(* CoDeSys 2.3.9.41 project: OWENProject.pro *)
(* Libraries: Util.lib 18.5.10 15:14:28, STANDARD.LIB 4.10.05 11:14:46, IECSFC.LIB 13.4.06 15:51:28, ANALYZATION.LIB 5.10.99 09:05:06 *)

(* PLC configuration (modules and I/O channels)
Fast discrete inputs [I_SIMPLE_INPUT] node 0, in %IB0 out %QB0 {Filtrationtime = 10}
  AT %IX0.0 [BitInput] Discrete input 1
  AT %IX0.1 [BitInput] Discrete input 2
  AT %IX0.2 [BitInput] Discrete input 3
  AT %IX0.3 [BitInput] Discrete input 4
Discrete inputs [ID130] node 1, in %IB1 out %QB1 {Filtrationtime_GeneralINP = 10; Visibility = No; PinCount = 12}
  AT %IB1.0 [ByteInput] 8 discrete inputs
  AT %IB1.1 [ByteInput] 4 discrete inputs
AT %QB2.0 [ByteOutput] 8 discrete outputs
AT %QB2.1 [ByteOutput] 4 discrete outputs
AT %IR3.0 [FloatInputP] AI #1 {AIN_TYPE = 4-20 mA; Peak_Filtr = 200; Flt_Ch = Off; TauRC = 10; MinFV = 0; MaxFV = 50}
AT %IR3.1 [FloatInputP] AI #2 {AIN_TYPE = 4-20 mA; Peak_Filtr = 200; Flt_Ch = Off; TauRC = 10; MinFV = 0; MaxFV = 50}
AT %IR3.2 [FloatInputP] AI #3 {AIN_TYPE = 4-20 mA; Peak_Filtr = 200; Flt_Ch = Off; TauRC = 10; MinFV = 0; MaxFV = 50}
AT %IR3.3 [FloatInputP] AI #4 {AIN_TYPE = 4-20 mA; Peak_Filtr = 200; Flt_Ch = Off; TauRC = 10; MinFV = 0; MaxFV = 20000.0}
AT %IR3.4 [FloatInputP] AI #5 {AIN_TYPE = 4-20 mA; Peak_Filtr = 200; Flt_Ch = Off; TauRC = 10; MinFV = 0; MaxFV = 20000.0}
AT %IR3.5 [FloatInputP] AI #6 {AIN_TYPE = 4-20 mA; Peak_Filtr = 200; Flt_Ch = Off; TauRC = 10; MinFV = 0; MaxFV = 20000.0}
AT %IR3.6 [FloatInputP] AI #7 {AIN_TYPE = 4-20 mA; Peak_Filtr = 200; Flt_Ch = Off; TauRC = 10; MinFV = 0; MaxFV = 20000.0}
AT %IR3.7 [FloatInputP] AI #8 {AIN_TYPE = 4-20 mA; Peak_Filtr = 200; Flt_Ch = Off; TauRC = 10; MinFV = 0; MaxFV = 20000.0}
AT %IW3.8 [WordInput] AI read time (10ms)
AT %QR4.0 [FloatOutputP] AO #1 {AOUT_TYPE = 0-10V; SafeValueREAL = 0.0}
AT %QR4.1 [FloatOutputP] AO #2 {AOUT_TYPE = 0-10V; SafeValueREAL = 0.0}
AT %QR4.2 [FloatOutputP] AO #3 {AOUT_TYPE = 0-10V; SafeValueREAL = 0.0}
AT %QR4.3 [FloatOutputP] AO #4 {AOUT_TYPE = 4-20 mA; SafeValueREAL = 0.0}
Special input [ID103] node 5, in %IB5 out %QB5 {Filtrationtime = 1000; PinCount = 1; WatchDogPeriod = 400; PollPeriod = 3000; Visibility = No}
  AT %IX5.0 [BitInput] Special input
Special output [ID104] node 6, in %IB6 out %QB6 {Visibility = No; PinCount = 1}
  AT %QX6.0 [BitOutput] Special output
Owen (Master) [OWEN_MASTER_ID451] node 7, in %IB7 out %QB7 {Timeout = 50; Visibility = Yes}
  AT %QW7.0 [WordOutput] Last error
  AT %QW7.1 [WordOutput] Last hash
  AT %QW7.2 [WordOutput] Last address
  AT %QB7.3 [ComChannel] Start/Stop)
  RS-485-1 [COM1_USART] node 0, in %IB7.0 out %QB7.0 {CommunicationSpeed = 9600; Parity = NO PARITY CHECK; BitLength = 8 bits; StopLength = One stop bit; InterfaceType = RS485; FrameOriented = ASCII; Timeout = 2; Visibility = No}
AT %QD7.1.0.0 [DWordOutput] MV110-32DN Digital Inputs
ModBus (Master) [MODBUS_MASTER_ID450] node 8, in %IB8 out %QB8 {Visibility = No}
  AT %QD8.0 [DWordOutput] Last address
  AT %QW8.1 [WordOutput] Last error
  RS-485-1 [COM1_USART] node 0, in %IB8.0 out %QB8.0 {CommunicationSpeed = 9600; Parity = NO PARITY CHECK; BitLength = 8 bits; StopLength = One stop bit; InterfaceType = RS485; FrameOriented = RTU; Timeout = 0; Visibility = No}
AT %QB8.1.0 [ComChannel] Command (0xff - Start)
AT %QW8.1.0.0 [WordOutput]
AT %QW8.1.1.0 [WordOutput]
AT %QW8.1.2.0 [WordOutput]
Value on output 4 [ID2085] node 3, in %IB8.1.3 out %QB8.1.3 {ModbusAddress = 3; Comm_Write_16 = Command Write (16); Visibility = No}
  AT %QW8.1.3.0 [WordOutput]
Value on output 5 [ID2086] node 4, in %IB8.1.4 out %QB8.1.4 {ModbusAddress = 4; Comm_Write_16 = Command Write (16); Visibility = No}
  AT %QW8.1.4.0 [WordOutput]
Value on output 6 [ID2087] node 5, in %IB8.1.5 out %QB8.1.5 {ModbusAddress = 5; Comm_Write_16 = Command Write (16); Visibility = No}
  AT %QW8.1.5.0 [WordOutput]
Value on output 7 [ID2088] node 6, in %IB8.1.6 out %QB8.1.6 {ModbusAddress = 6; Comm_Write_16 = Command Write (16); Visibility = No}
  AT %QW8.1.6.0 [WordOutput]
Value on output 8 [ID2089] node 7, in %IB8.1.7 out %QB8.1.7 {ModbusAddress = 7; Comm_Write_16 = Command Write (16); Visibility = No}
  AT %QW8.1.7.0 [WordOutput]
PWM period on output 1 [ID2090] node 8, in %IB8.1.8 out %QB8.1.8 {ModbusAddress = 32; Comm_Write_16 = Command Write (16); Visibility = No}
  AT %QW8.1.8.0 [WordOutput]
PWM period on output 2 [ID2091] node 9, in %IB8.1.9 out %QB8.1.9 {ModbusAddress = 33; Comm_Write_16 = Command Write (16); Visibility = No}
  AT %QW8.1.9.0 [WordOutput]
PWM period on output 3 [ID2092] node 10, in %IB8.1.10 out %QB8.1.10 {ModbusAddress = 34; Comm_Write_16 = Command Write (16); Visibility = No}
  AT %QW8.1.10.0 [WordOutput]
PWM period on output 4 [ID2093] node 11, in %IB8.1.11 out %QB8.1.11 {ModbusAddress = 35; Comm_Write_16 = Command Write (16); Visibility = No}
  AT %QW8.1.11.0 [WordOutput]
PWM period on output 5 [ID2094] node 12, in %IB8.1.12 out %QB8.1.12 {ModbusAddress = 36; Comm_Write_16 = Command Write (16); Visibility = No}
  AT %QW8.1.12.0 [WordOutput]
PWM period on output 6 [ID2095] node 13, in %IB8.1.13 out %QB8.1.13 {ModbusAddress = 37; Comm_Write_16 = Command Write (16); Visibility = No}
  AT %QW8.1.13.0 [WordOutput]
PWM period on output 7 [ID2096] node 14, in %IB8.1.14 out %QB8.1.14 {ModbusAddress = 38; Comm_Write_16 = Command Write (16); Visibility = No}
  AT %QW8.1.14.0 [WordOutput]
PWM period on output 8 [ID2097] node 15, in %IB8.1.15 out %QB8.1.15 {ModbusAddress = 39; Comm_Write_16 = Command Write (16); Visibility = No}
  AT %QW8.1.15.0 [WordOutput]
*)

(* Task configuration *)
TASK TaskFreewheeling (PRIORITY := 1); (* freewheeling *)
	PLC_PRG();
END_TASK
TASK Task200ms (PRIORITY := 1, INTERVAL := T#200ms);
	GetInputs();
END_TASK
TASK Task1Sec (PRIORITY := 1, INTERVAL := T#1000ms);
	SetOutputs();
END_TASK

(* Global variable list: Global_Variables *)
VAR_GLOBAL CONSTANT
	MAXIMUM_HEATING_CIRCUITS_NUM : USINT := 3;
	(*Количество отопительных контуров*)

	MAX_UZ_NUM : USINT := 3;
	(*Количество частотных преобразователей UZ*)

	MAX_BOILERS_NUM : USINT := 3;
	(*Количество котлов*)

	MAX_K14_PUMPS_NUM : USINT := 3;
	(*Количество насосов К14*)

	MAX_K15_PUMPS_NUM : USINT := 2;
	(*Количество насосов К15*)

	MAX_K16_PUMPS_NUM : USINT := 2;
	(*Количество насосов К16*)
END_VAR

VAR_GLOBAL
	PLC160DI : strPLC160DI;
	PLC160AI : strPLC160AI;
	PLC160DO : strPLC160DO;
	PLC160AO : strPLC160AO;
	MV110DI  : strMV110DI;
	MU110DO  : strMU110DO;

	K14PumpFaulty : ARRAY [1..MAX_K14_PUMPS_NUM] OF BOOL;
	(*Неиправен 1-3 насос группы К14?*)

	K15PumpFaulty : ARRAY [1..MAX_K15_PUMPS_NUM] OF BOOL;
	(*Неиправен 1-3 насос группы К16?*)

	K16PumpFaulty : ARRAY [1..MAX_K16_PUMPS_NUM] OF BOOL;
	(*Неиправен 1-3 насос группы К16?*)
END_VAR

(* Global variable list: PLC_IO *)
VAR_GLOBAL
(* Дискретные входы ПЛК160*)
	DI_0_00  AT %IX0.0 : BOOL;
	DI_0_01  AT %IX0.1 : BOOL;
	DI_0_02  AT %IX0.2 : BOOL;
	DI_0_03  AT %IX0.3 : BOOL;
	DI_0_04  AT %IX1.0.0 : BOOL;
	DI_0_05  AT %IX1.0.1 : BOOL;
	DI_0_06  AT %IX1.0.2 : BOOL;
	DI_0_07  AT %IX1.0.3 : BOOL;
	DI_0_08  AT %IX1.0.4 : BOOL;
	DI_0_09  AT %IX1.0.5 : BOOL;
	DI_0_10  AT %IX1.0.6 : BOOL;
	DI_0_11  AT %IX1.0.7 : BOOL;
	DI_0_12  AT %IX1.1.0 : BOOL;
	DI_0_13  AT %IX1.1.1 : BOOL;
	DI_0_14  AT %IX1.1.2 : BOOL;
	DI_0_15  AT %IX1.1.3 : BOOL;

(* Аналоговые входы ПЛК160*)
	AI_0_00 AT %IR3.0 : REAL;
	AI_0_01 AT %IR3.1 : REAL;
	AI_0_02 AT %IR3.2 : REAL;
	AI_0_03 AT %IR3.3 : REAL;
	AI_0_04 AT %IR3.4 : REAL;
	AI_0_05 AT %IR3.5 : REAL;
	AI_0_06 AT %IR3.6 : REAL;
	AI_0_07 AT %IR3.7 : REAL;

(*Аналоговые выходы ПЛК160*)
	AO_0_00 AT %QR4.0 : REAL;
	AO_0_01 AT %QR4.1 : REAL;
	AO_0_02 AT %QR4.2 : REAL;
	AO_0_03 AT %QR4.3 : REAL;

(*Дискретные выходы ПЛК160*)
	DO_0_00 AT %QX2.0.0 : BOOL;
	DO_0_01 AT %QX2.0.1 : BOOL;
	DO_0_02 AT %QX2.0.2 : BOOL;
	DO_0_03 AT %QX2.0.3 : BOOL;
	DO_0_04 AT %QX2.0.4 : BOOL;
	DO_0_05 AT %QX2.0.5 : BOOL;
	DO_0_06 AT %QX2.0.6 : BOOL;
	DO_0_07 AT %QX2.0.7 : BOOL;

	DO_0_08 AT %QX2.1.0 : BOOL;
	DO_0_09 AT %QX2.1.1 : BOOL;
	DO_0_10 AT %QX2.1.2 : BOOL;
	DO_0_11 AT %QX2.1.3 : BOOL;

(*Дискретные входы МВ110-32ДН*)
	DI_1 AT %QD7.1.0.0 : DWORD;

(*Дискретные выходы МУ110-8Р*)
	DO_1_00 AT %QW8.1.0.0 : WORD;
	DO_1_01 AT %QW8.1.1.0 : WORD;
	DO_1_02 AT %QW8.1.2.0 : WORD;
	DO_1_03 AT %QW8.1.3.0 : WORD;
	DO_1_04 AT %QW8.1.4.0 : WORD;
	DO_1_05 AT %QW8.1.5.0 : WORD;
	DO_1_06 AT %QW8.1.6.0 : WORD;
	DO_1_07 AT %QW8.1.7.0 : WORD;


END_VAR

(* Global variable list: Variable_Configuration *)
VAR_GLOBAL RETAIN
	K14UZSPumpSpeed : USINT := 100;
END_VAR

(* Data type *)
TYPE strMU110DO :
STRUCT
	K14PumpGroupAlarm : BOOL;
(*
	Выход №1
	Авария насосной группы К14
*)

	Buzzer : BOOL;
(*
	Выход №2
	Зуммер
*)

	K14PumpIsOn : ARRAY [1..MAX_K14_PUMPS_NUM] OF BOOL;
(*
	Выходы №3-5
	"Насос К14.1-3 в работе"
*)

	Reserved : ARRAY [1..3] OF BOOL;
(*
	Выходы 6-8
	Резерв
*)


END_STRUCT
END_TYPE

(* Data type *)
TYPE strMV110DI :
(*
	поз. А2
	Контроллер МВ110-32 ДН
	Дискретные входы
*)
STRUCT
	K15_StopButton : ARRAY [1..2] OF BOOL;
(*
	Входы №1-2
	Сигналы с кнопок стоп Насосов К15.1-2
*)

	K16_StopButton : ARRAY [1..2] OF BOOL;
(*
	Входы №3-4
	Сигналы с кнопок стоп Насосов К16.1-2
*)

	K15_NoPressureDrop : BOOL;
(*
	Вход №5
	Сигнал с датчика перепада давления
	"Нет перепада давления на насосной группе К15"
	Замкнут - "Нет перепада".
*)

	K16_NoPressureDrop : BOOL;
(*
	Вход №6
	Сигнал с датчика перепада давления
	"Нет перепада давления на насосной группе К16"
	Замкнут - "Нет перепада".
*)

	HeatingDHWPumpGroupModeIsAuto : BOOL;
(*
	Вход №7
	Сигнал переключателя "Работа в автоматическом режиме
	насосной группы К15 греющего контура ГВС"
*)

	DHWPumpGroupModeIsAuto : BOOL;
(*
	Вход №8
	Сигнал переключателя "Работа в автоматическом режиме
	насосной группы К16 контура ГВС"
*)

	CO_Level_I : BOOL;
(*
	Вход №9
	I уровень загазованности по CO
*)

	CO_Level_II : BOOL;
(*
	Вход №10
	II уровень загазованности по CO
*)

	CH_Level_I : BOOL;
(*
	Вход №11
	I уровень загазованности по CH
*)

	CH_Level_II : BOOL;
(*
	Вход №12
	II уровень загазованности по CH
*)

	FireAlarm : BOOL;
(*
	Вход №13
	Пожар в энергоцентре
*)

	BoilerGeneralFault : BOOL;
(*
	Вход №14
	Сигнал с панели управления котлов ведущей ПУКВ
	"Общая неисправность котлов"
*)

	TurnOnK15AndK16 : BOOL;
(*
	Вход №15
	Сигнал с панели управления котлов ведущей ПУКВ,
	"Включить/Выключить насосную группу К15 и К16"
*)

	K22ValveState : strValveState;
(*
	Входы №16-17
	Сигналы положения 3-х ходового клапана К22 "Открыт"/"Закрыт"
*)

	K23ValveState : strValveState;
(*
	Входы №18-19
	Сигналы положения 3-х ходового клапана К23 "Открыт"/"Закрыт"
*)

	BoilerAlarm : ARRAY [1..MAX_BOILERS_NUM] OF BOOL;
(*
	Входы №20-22
	Сигналы с ЩАК1-3 "Авария котла №1-3"
*)

	BlockAllBoilers : BOOL;
(*
	Вход №23
	Блокировка всех котлов
*)

	TurnOnAllBoilers : BOOL;
(*
	Вход №24
	Сигнал внешнего включения всех котлов
*)

	SignalizationButton : BOOL;
(*
	Вход №25
	Кнопка съема сигнализации
*)

	QFSwitcher : ARRAY [1..7] OF BOOL;
(*
	Входы №26-32
	Доп. контакты автоматических выключателей QF1-7
	1-3 Включение/выключение частотных модуляторов UZ
	4-5 - Включение/выключение насосов К15
	6-7 - Включение/выключение насосов К16
*)


END_STRUCT
END_TYPE

(* Data type *)
TYPE strPLC160AI :
(*
	поз. А1
	Контроллер ПЛК160
	Аналоговые входы
*)
STRUCT
	UZSignal : ARRAY [1..MAX_UZ_NUM] OF tUZSignal;
(*
	Аналоговые входы №1-3:
	Сигналы 0-20mA от частотных преобразователей UZ
*)

	DilutionSignal : ARRAY [1..MAX_BOILERS_NUM] OF tDelutionSignal;
(*
	Аналоговые входы №4-6:
	Сигналы 4-20mA измерения разрежения из щита ЩИР
	по одному сигналу на каждый котел
*)

	Reserved : ARRAY [1..2] OF tAnalogInput;
(*
	Незадействованные входы
*)


END_STRUCT
END_TYPE

(* Data type *)
(*
	поз. А1
	Контроллер ПЛК160
	Аналоговые выходы
*)
TYPE strPLC160AO :
STRUCT
(*
	Выходы №1-3
	Задание частоты для UZ1-3
	Сигнал 0-10V
*)
	UZSpeed : ARRAY [1..MAX_UZ_NUM] OF tUZSpeed;

(*
	Выход №4
	Резерв
*)
	Reserved : tAnalogOutput;
END_STRUCT
END_TYPE

(* Data type *)
TYPE strPLC160DI :
STRUCT
	K14_PumpsModeIsAuto : BOOL;
(*
	Дискретных вход №1:
	Сигнал с переключателя режима работы насосов К14
	"Ручной/Автоматический". Замкнут - "Автоматический"
*)

	K14_PumpsModeIsHeating : BOOL;
(*
	Дискретный вход №2:
	Сигнал с переключателя режима работы насосов К14
	"Летний/Отопительный". Замкнут - "Отопительный"
*)

	K14_PumpStop : ARRAY [1..MAX_K14_PUMPS_NUM] OF BOOL;
(*
	Дискретный вход №3-5:
	Сигнал с кнопки "Стоп насос К14.1-3".
	Замкнут - "Кнопка нажата".
	Аварийный СТОП насоса
*)

	K14_NoPressureDrop : BOOL;
(*
	Дискретный вход №6:
	Сигнал с датчика перепада давления
	насосной группы К14.
	Замкнут - нет перепада.
*)

	UZStatus : ARRAY [1..MAX_UZ_NUM] OF strUZStatus;
(*
	Дискретные входы №7-15:
	Сигналы част. преобр. UZ1-UZ3
*)

	Reserved : BOOL;
(*
	Дискретный вход №16:
	Резерв
*)


END_STRUCT
END_TYPE

(* Data type *)
TYPE strPLC160DO :
(*
	поз. А1
	Контроллер ПЛК160
	Дискретные выходы
*)
STRUCT
	UZStart : ARRAY [1..MAX_UZ_NUM] OF BOOL;
(*
	Выходы №1-3
	Пуск UZ
*)

	UZConstSpeed : ARRAY [1..MAX_UZ_NUM] OF BOOL;
(*
	Выходы №4-6
	Выбор постоянной скорости UZ (50Гц, 100%)
*)

	K15Pump : ARRAY [1..2] OF BOOL;
(*
	Выходы №7-8
	Включить/отключить насосы К15.1-2
*)

	K16Pump : ARRAY [1..2] OF BOOL;
(*
	Выходы №9-10
	Включить/отключить насосы К16.1-2
*)

	K15Alarm : BOOL;
(*
	Выход №11
	Авария насосной группы К15
*)

	K16Alarm : BOOL;
(*
	Выход №12
	Авария насосной группы К16
*)



END_STRUCT
END_TYPE

(* Data type *)
(*Сигналы с част. преобр UZ*)
TYPE strUZStatus :
STRUCT
	Ready : BOOL;
	Running : BOOL;
	Fail	: BOOL;
END_STRUCT
END_TYPE

(* Data type *)
(*Состояние 3-х ходового клапана*)
TYPE strValveState :
STRUCT
	Open : BOOL;
	Close: BOOL;
END_STRUCT
END_TYPE

(* Data type *)
TYPE tAnalogInput : REAL;
END_TYPE

(* Data type *)
TYPE tAnalogOutput : REAL;
END_TYPE

(* Data type *)
TYPE tDelutionSignal : REAL;
END_TYPE

(* Data type *)
TYPE tUZSignal : REAL;
END_TYPE

(* Data type *)
TYPE tUZSpeed : REAL;
END_TYPE

(* POU PLC_PRG, ST *)
PROGRAM PLC_PRG
VAR CONSTANT
	K14AutoModeDelay : TIME := T#10s;
END_VAR

VAR
	SignalizationResetTrigger : F_TRIG;
	K14PumpsControl : fbK14PumpsControl;
	K15PumpsControl : fbK15PumpsControl;
	K16PumpsControl : fbK16PumpsControl;
	K14ManualModeTOF : TOF;
END_VAR

VAR_TEMP
	i: USINT;
	K14WorkAllowed : BOOL := FALSE;

	K15WorkAllowed: BOOL := FALSE;

	K16WorkAllowed : BOOL := FALSE;
END_VAR
	K14WorkAllowed := FALSE;

	K15WorkAllowed := FALSE;

	K16WorkAllowed := FALSE;

(*
	Проверить состояние аварий на насосах и зажечь лампочки, включить зуммер
*)
checkPumpsAlarm();

(*
	Проверить состояние всех других аварий и включить зуммер
*)
checkOtherAlarms();

(*
	Сброс всех аварий насосов по замыканию кнопки
	съема аварий
*)
SignalizationResetTrigger(CLK := MV110DI.SignalizationButton);
resetPumpsAlarm(SignalizationResetTrigger.Q);


(*
	Включение сигнала на UZ
	по тому же сигналу, что и MV110DI.TurnOnK15AndK16
FOR i := 1 TO MAX_K14_PUMPS_NUM DO
	PLC160DO.UZStart[i] := MV110DI.TurnOnK15AndK16;
END_FOR;
*)

(*
	3. Управление насосами К14
	контура отопления и вентиляции
*)
FOR i := 1 TO MAX_K14_PUMPS_NUM DO
	MU110DO.K14PumpIsOn[i] := PLC160DI.UZStatus[i].Running;
	(*Включить/Выключить сигнальную лампу состояния насоса*)

	(*если хоть один из насосов исправен, то работа разрешена*)
	IF NOT(K14PumpFaulty[i]) THEN
		K14WorkAllowed := TRUE;
	END_IF;
END_FOR;

K14ManualModeTOF(IN := NOT(PLC160DI.K14_PumpsModeIsAuto), PT := K14AutoModeDelay);

K14PumpsControl(
	ManualMode						:= K14ManualModeTOF.Q,
	WorkAllowed						:= K14WorkAllowed,
	SummerMode						:= NOT(PLC160DI.K14_PumpsModeIsHeating),
	EmergencyPumpStopButtonPressed := PLC160DI.K14_PumpStop,
	PumpState						:= MU110DO.K14PumpIsOn,
	PressureDrop					:= NOT(PLC160DI.K14_NoPressureDrop)
);

(*
	6. Управление насосами К15
	греющего контура ГВС
*)
FOR i := 1 TO MAX_K15_PUMPS_NUM DO
	(*если хоть один из насосов исправен, то работа разрешена*)
	IF NOT(K15PumpFaulty[i]) THEN
		K15WorkAllowed := TRUE;
	END_IF;
END_FOR;

K15PumpsControl(
	ManualMode						:= NOT(MV110DI.HeatingDHWPumpGroupModeIsAuto),
	WorkAllowed						:= K15WorkAllowed,
	EmergencyPumpStopButtonPressed := MV110DI.K15_StopButton,
	PumpState						:= PLC160DO.K15Pump,
	PressureDrop					:= NOT(MV110DI.K15_NoPressureDrop)
);

(*
	5. Управление насосами К16
	контура ГВС
*)
FOR i := 1 TO MAX_K16_PUMPS_NUM DO
	(*если хоть один из насосов исправен, то работа разрешена*)
	IF NOT(K16PumpFaulty[i]) THEN
		K16WorkAllowed := TRUE;
	END_IF;
END_FOR;

K16PumpsControl(
	ManualMode						:= NOT(MV110DI.DHWPumpGroupModeIsAuto),
	WorkAllowed						:= K16WorkAllowed,
	EmergencyPumpStopButtonPressed := MV110DI.K16_StopButton,
	PumpState						:= PLC160DO.K16Pump,
	PressureDrop					:= NOT(MV110DI.K16_NoPressureDrop)
);
END_PROGRAM

(* POU K14/fbK14PumpsControl, ST *)
FUNCTION_BLOCK fbK14PumpsControl
(*
	3. Управление насосами К14
	контура отопления и вентиляции
*)
VAR CONSTANT
	PumpCheckDelayTime : TIME := T#30s;
END_VAR

VAR_INPUT
	ManualMode: BOOL;						(*Ручной режим?*)
	WorkAllowed: BOOL;					(*Работа разрешена?*)
	SummerMode: BOOL;						(*Летний режим?*)
	EmergencyPumpStopButtonPressed: ARRAY [1..MAX_K14_PUMPS_NUM] OF BOOL; (*Нажат аварийный стоп насоса?*)
	PumpState: ARRAY [1..MAX_K14_PUMPS_NUM] OF BOOL;	(*Работает насос?*)
	PressureDrop : BOOL;					(*Есть разница давлений?*)
END_VAR
VAR
	pumpStatusCheckDelay	: ARRAY [1..MAX_K14_PUMPS_NUM] OF TON;
	workOrderControl : fbK14WorkOrderControl;
	pumpsTrainingControl : fbK14PumpsTraining;
END_VAR
VAR_TEMP
	i: USINT;
	pumpWorkOrder : ARRAY [1..MAX_K14_PUMPS_NUM] OF USINT;
	pumpStatusCheck : ARRAY [1..MAX_K14_PUMPS_NUM] OF BOOL;
	break : BOOL := FALSE;
END_VAR
break := FALSE;
(*Проверяем исправность насосов К14*)
FOR i := 1 TO MAX_K14_PUMPS_NUM DO
	pumpStatusCheckDelay[i](IN := PumpState[i], PT := PumpCheckDelayTime);
	pumpStatusCheck[i] := pumpStatusCheckDelay[i].Q;
END_FOR;

fK14PumpsFaultyControl(
	PumpState				:= PumpState,
	PumpStatusCheckDelay	:= pumpStatusCheck,
	PressureDrop			:= PressureDrop
);

(*Управление насосами К14*)
IF ManualMode THEN (*Ручной режим?*)
(*
	FOR i := 1 TO MAX_K14_PUMPS_NUM DO
		fK14PumpManualControl(
			PumpID	:= i,
			TurnOn	:= TurnOnPumpButtonPressed[i],
			TurnOff	:= TurnOffPumpButtonPressed[i],
			State		:= PumpState[i],
			EmergencyStop := EmergencyPumpStopButtonPressed[i]
		);
	END_FOR;
*)
	(*Контроллер никак не участвует в ручном режиме*)
	FOR i := 1 TO MAX_K14_PUMPS_NUM DO
		fTurnOffK14Pump(i);
	END_FOR;
ELSE
	IF WorkAllowed THEN	(*Работа разрешена?*)
		(*определяем порядок включения насосов*)
		workOrderControl( SummerMode := SummerMode,
								pumpWorkOrder := pumpWorkOrder);

		FOR i := 1 TO MAX_K14_PUMPS_NUM DO
			(*
				работаем с насосами в порядке их приоритета
				Ищем первый исправный насос и включаем его
			*)
			IF NOT(break) AND NOT(K14PumpFaulty[pumpWorkOrder[i]]) THEN
				fK14PumpAutoControl(
						PumpID := pumpWorkOrder[i],
						EmergencyPumpStopButtonPressed := EmergencyPumpStopButtonPressed[pumpWorkOrder[i]]
				);
				break := TRUE;
			END_IF;
		END_FOR;
		(*периодическая тренировка насосов*)
		pumpsTrainingControl();
	ELSE
		(*
			если работа не разрешена,
			выключаем все насосы
		*)
		FOR i := 1 TO MAX_K14_PUMPS_NUM DO
			fTurnOffK14Pump(i);
		END_FOR;
		RETURN;
	END_IF;
END_IF;
END_FUNCTION_BLOCK

(* POU K14/fbK14WorkOrderControl, ST *)
FUNCTION_BLOCK fbK14WorkOrderControl
VAR_INPUT
	SummerMode: BOOL;
END_VAR

VAR CONSTANT
	MAX_K14_HEATING_ORDERS_NUM : USINT := 2;
	PumpWorkSummerOrder : ARRAY [1..MAX_K14_PUMPS_NUM] OF USINT := 3, 1, 2;
	PumpWorkHeatingOrder : ARRAY [1..MAX_K14_HEATING_ORDERS_NUM,
											1..MAX_K14_PUMPS_NUM] OF USINT := 1, 2, 3, 2, 1, 3;
END_VAR
VAR
	workOrderChanger		: BLINK;
	K14PumpsHeatingWorkOrderID : USINT(1..MAX_K14_HEATING_ORDERS_NUM) := 1;
END_VAR
VAR_IN_OUT
	pumpWorkOrder : ARRAY [1..MAX_K14_PUMPS_NUM] OF USINT;
END_VAR
VAR_TEMP
	i: USINT;
END_VAR
IF SummerMode THEN	(*Летний режим?*)
	pumpWorkOrder := PumpWorkSummerOrder;
ELSE

	workOrderChanger(
		ENABLE := TRUE,
		TIMELOW := T#24h,
		TIMEHIGH := T#24h
	);

	IF workOrderChanger.OUT THEN
		K14PumpsHeatingWorkOrderID := 1;
	ELSE
		K14PumpsHeatingWorkOrderID := 2;
	END_IF;

	FOR i := 1 TO MAX_K14_PUMPS_NUM DO
		pumpWorkOrder[i] := PumpWorkHeatingOrder[K14PumpsHeatingWorkOrderID, i];
	END_FOR;
END_IF;
END_FUNCTION_BLOCK

(* POU K14/fbK14PumpsTraining, ST *)
FUNCTION_BLOCK fbK14PumpsTraining
(*
	Функция тренировки насосов К14
*)
VAR CONSTANT
	TrainingDelay: TIME := T#24h;		(*Задержка на включение тренировки*)
	TrainingPeriod: TIME := T#10s;	(*Период тренировки*)
END_VAR
VAR
	PumpOffDelay : ARRAY [1..MAX_K14_PUMPS_NUM] OF TON;
	PumpTrainingTimer : ARRAY [1..MAX_K14_PUMPS_NUM] OF TP;
END_VAR
VAR_TEMP
	i: USINT;
END_VAR
FOR i := 1 TO MAX_K14_PUMPS_NUM DO
	PumpOffDelay[i](IN := fGetK14Pump(i), PT := TrainingDelay);
	PumpTrainingTimer[i](IN := PumpOffDelay[i].Q, PT := TrainingPeriod);
	IF PumpTrainingTimer[i].Q THEN
		fTurnOnK14Pump(i);
	END_IF;
END_FOR;
END_FUNCTION_BLOCK

(* POU K14/fGetK14Pump, ST *)
FUNCTION fGetK14Pump :BOOL
(* Проверка включения насоса*)
VAR_INPUT
	PumpID : USINT;
END_VAR
fGetK14Pump := MU110DO.K14PumpIsOn[PumpID];
END_FUNCTION

(* POU K14/fTurnOnK14Pump, ST *)
FUNCTION fTurnOnK14Pump : BOOL
VAR_INPUT
	PumpID : USINT;
END_VAR
VAR
END_VAR
	fSetK14Pump(TRUE, PumpID);
END_FUNCTION

(* POU K14/fSetK14Pump, ST *)
FUNCTION fSetK14Pump : BOOL
VAR_INPUT
	State	: BOOL;
	PumpID : USINT;
END_VAR
VAR
END_VAR
	(*Задать управляющее напряжение на насос*)
	IF State THEN
		PLC160DO.UZStart[PumpID]		:= TRUE;
		PLC160AO.UZSpeed[PumpID]	:= fUZSignalToVoltageOutput(K14UZSPumpSpeed);
	ELSE
		PLC160DO.UZStart[PumpID]		:= FALSE;
		PLC160AO.UZSpeed[PumpID]	:= 0.0;
	END_IF;
END_FUNCTION

(* POU K14/fUZSignalToVoltageOutput, ST *)
FUNCTION fUZSignalToVoltageOutput : REAL
(*
	Функция преобразования входного
	сигнала 0-100% в выходное управляющее
	напряжение на насос
*)
VAR_INPUT
	IN : USINT; (*Входной сигнал*)
END_VAR
VAR
END_VAR
(*TODO: написать корректную функцию преобразования тока в напряжение*)
fUZSignalToVoltageOutput := IN/10.0;
END_FUNCTION

(* POU K14/fK14PumpsFaultyControl, ST *)
FUNCTION fK14PumpsFaultyControl : BOOL
(* Проверка состояния насосов*)
VAR_INPUT
	PumpState : ARRAY [1..MAX_K14_PUMPS_NUM] OF BOOL;
	PumpStatusCheckDelay : ARRAY [1..MAX_K14_PUMPS_NUM] OF BOOL;
	PressureDrop : BOOL;
END_VAR
VAR
	i : USINT;
	activePumpID : USINT; (*номер работающего насоса*)
END_VAR
activePumpID := 0;

FOR i := 1 TO MAX_K14_PUMPS_NUM DO
	IF PumpState[i] THEN
		IF activePumpID <> 0 THEN
			(*
				Включено больше одного насоса -
				ничего не можем сказать об их исправности
			*)
			RETURN;
		END_IF;
		activePumpID := i;
	END_IF;
END_FOR;

IF activePumpID = 0 THEN
	(*
		Не включен ни один насос - 
		ничего не можем сказать об их исправности
	*)
	RETURN;
END_IF;

IF PumpStatusCheckDelay[activePumpID] THEN
	(*
		Определяем исправность насоса
		по перепаду давления
	*)
	K14PumpFaulty[activePumpID] := NOT(PressureDrop);
END_IF;
END_FUNCTION

(* POU K14/fTurnOffK14Pump, ST *)
FUNCTION fTurnOffK14Pump : BOOL
VAR_INPUT
	PumpID : USINT;
END_VAR
VAR
END_VAR
	fSetK14Pump(FALSE, PumpID);
END_FUNCTION

(* POU K14/fK14PumpAutoControl, ST *)
FUNCTION fK14PumpAutoControl : BOOL
VAR_INPUT
	PumpID : USINT;
	EmergencyPumpStopButtonPressed : BOOL;
END_VAR
VAR
	i : USINT;
END_VAR
(*выключаем все насосы кроме данного*)
FOR i := 1 TO MAX_K14_PUMPS_NUM DO
	IF i <> PumpID THEN
		fTurnOffK14Pump(i);
	END_IF;
END_FOR;

IF EmergencyPumpStopButtonPressed THEN	(*Нажат аварийный стоп насоса?*)
	fTurnOffK14Pump(PumpID); (*Выключить насос*)
	RETURN;
END_IF;

IF K14PumpFaulty[PumpID] THEN
	fTurnOffK14Pump(PumpID); (*Выключить насос*)
ELSE
	fTurnOnK14Pump(PumpID); (*Включить насос*)
END_IF;
END_FUNCTION

(* POU K15/fbK15PumpsControl, ST *)
FUNCTION_BLOCK fbK15PumpsControl
(*
	Управление насосами К15
	контура нагрева ГВС
*)
VAR CONSTANT
	PumpCheckDelayTime : TIME := T#10s;
	PumpWorkHeatingOrder : ARRAY [1..MAX_K15_PUMPS_NUM] OF USINT := 1, 2;
END_VAR
VAR_INPUT
	ManualMode: BOOL;						(*Ручной режим?*)
	WorkAllowed: BOOL;					(*Работа разрешена?*)
	EmergencyPumpStopButtonPressed: ARRAY [1..MAX_K15_PUMPS_NUM] OF BOOL; (*Нажат аварийный стоп насоса?*)
	PumpState: ARRAY [1..MAX_K15_PUMPS_NUM] OF BOOL;	(*Работает насос?*)
	PressureDrop : BOOL;					(*Есть разница давлений?*)
END_VAR
VAR_OUTPUT
END_VAR
VAR
	pumpStatusCheckDelay	: ARRAY [1..MAX_K15_PUMPS_NUM] OF TON;
	pumpsTrainingControl : fbK15PumpsTraining;
END_VAR

VAR_TEMP
	i : USINT;
	pumpWorkOrder : ARRAY [1..MAX_K15_PUMPS_NUM] OF USINT;
	pumpStatusCheck : ARRAY [1..MAX_K15_PUMPS_NUM] OF BOOL;
	break : BOOL := FALSE;
END_VAR
break := FALSE;

FOR i := 1 TO MAX_K15_PUMPS_NUM DO
	pumpStatusCheckDelay[i](IN := PumpState[i], PT := PumpCheckDelayTime);
	pumpStatusCheck[i] := pumpStatusCheckDelay[i].Q;
END_FOR;

fK15PumpsFaultyControl(
	PumpState				:= PumpState,
	PumpStatusCheckDelay	:= pumpStatusCheck,
	PressureDrop			:= PressureDrop
);

IF ManualMode THEN (*Ручной режим?*)
(*
	FOR i := 1 TO MAX_K15_PUMPS_NUM DO
		fK15PumpManualControl(
			PumpID	:= i,
			TurnOn	:= TurnOnPumpButtonPressed[i],
			TurnOff	:= TurnOffPumpButtonPressed[i],
			State		:= PumpState[i],
			EmergencyStop := EmergencyPumpStopButtonPressed[i]
		);
	END_FOR;
*)
	(*Контроллер никак не участвует в ручном режиме*)
	FOR i := 1 TO MAX_K15_PUMPS_NUM DO
		fTurnOffK15Pump(i);
	END_FOR;
ELSE
	IF WorkAllowed THEN	(*Работа разрешена?*)
		pumpWorkOrder := PumpWorkHeatingOrder;
		FOR i := 1 TO MAX_K15_PUMPS_NUM DO
			(*
				работаем с насосами в порядке их приоритета
				Ищем первый исправный насос и включаем его
			*)
			IF NOT(break) AND NOT(K15PumpFaulty[pumpWorkOrder[i]]) THEN
				fK15PumpAutoControl(
						PumpID := pumpWorkOrder[i],
						EmergencyPumpStopButtonPressed := EmergencyPumpStopButtonPressed[pumpWorkOrder[i]]
				);
				break := TRUE;
			END_IF;
		END_FOR;
			(*периодическая тренировка насосов*)
		pumpsTrainingControl();
	ELSE
		(*
			если работа не разрешена,
			выключаем все насосы
		*)
		FOR i := 1 TO MAX_K15_PUMPS_NUM DO
			fTurnOffK15Pump(i);
		END_FOR;
		RETURN;
	END_IF;
END_IF;
END_FUNCTION_BLOCK

(* POU K15/fbK15PumpsTraining, ST *)
FUNCTION_BLOCK fbK15PumpsTraining
(*
	Функция тренировки насосов К15
*)
VAR CONSTANT
	TrainingDelay: TIME := T#24h;		(*Задержка на включение тренировки*)
	TrainingPeriod: TIME := T#10s;	(*Период тренировки*)
END_VAR
VAR
	PumpOffDelay : ARRAY [1..MAX_K15_PUMPS_NUM] OF TON;
	PumpTrainingTimer : ARRAY [1..MAX_K15_PUMPS_NUM] OF TP;
END_VAR
VAR_TEMP
	i: USINT;
END_VAR
FOR i := 1 TO MAX_K15_PUMPS_NUM DO
	PumpOffDelay[i](IN := fGetK15Pump(i), PT := TrainingDelay);
	PumpTrainingTimer[i](IN := PumpOffDelay[i].Q, PT := TrainingPeriod);
	IF PumpTrainingTimer[i].Q THEN
		fTurnOnK15Pump(i);
	END_IF;
END_FOR;
END_FUNCTION_BLOCK

(* POU K15/fGetK15Pump, ST *)
FUNCTION fGetK15Pump :BOOL
(* Проверка включения насоса*)
VAR_INPUT
	PumpID : USINT;
END_VAR
fGetK15Pump := PLC160DO.K15Pump[PumpID];
END_FUNCTION

(* POU K15/fTurnOnK15Pump, ST *)
FUNCTION fTurnOnK15Pump :BOOL
VAR_INPUT
	PumpID : USINT;
END_VAR
VAR
END_VAR
fSetK15Pump(TRUE, PumpID);
END_FUNCTION

(* POU K15/fSetK15Pump, ST *)
FUNCTION fSetK15Pump : BOOL
VAR_INPUT
	State : BOOL;
	PumpID : USINT;
END_VAR
VAR
END_VAR
	PLC160DO.K15Pump[PumpID] := State;
	(*Включить/Выключить реле насоса*)
END_FUNCTION

(* POU K15/fK15PumpsFaultyControl, ST *)
FUNCTION fK15PumpsFaultyControl :BOOL
(* Проверка состояния насосов*)
VAR_INPUT
	PumpState : ARRAY [1..MAX_K15_PUMPS_NUM] OF BOOL;
	PumpStatusCheckDelay : ARRAY [1..MAX_K15_PUMPS_NUM] OF BOOL;
	PressureDrop : BOOL;
END_VAR
VAR
	i : USINT;
	activePumpID : USINT; (*номер работающего насоса*)
END_VAR
activePumpID := 0;

FOR i := 1 TO MAX_K15_PUMPS_NUM DO
	IF PumpState[i] THEN
		IF activePumpID <> 0 THEN
			(*
				Включено больше одного насоса -
				ничего не можем сказать об их исправности
			*)
			RETURN;
		END_IF;
		activePumpID := i;
	END_IF;
END_FOR;

IF activePumpID = 0 THEN
	(*
		Не включен ни один насос - 
		ничего не можем сказать об их исправности
	*)
	RETURN;
END_IF;

IF PumpStatusCheckDelay[activePumpID] THEN
	(*
		Определяем исправность насоса
		по перепаду давления
	*)
	K15PumpFaulty[activePumpID] := NOT(PressureDrop);
END_IF;
END_FUNCTION

(* POU K15/fTurnOffK15Pump, ST *)
FUNCTION fTurnOffK15Pump :BOOL
VAR_INPUT
	PumpID : USINT;
END_VAR
VAR
END_VAR
	fSetK15Pump(FALSE, PumpID);
END_FUNCTION

(* POU K15/fK15PumpAutoControl, ST *)
FUNCTION fK15PumpAutoControl :BOOL
VAR_INPUT
	PumpID : USINT;
	EmergencyPumpStopButtonPressed : BOOL;
END_VAR
VAR
	i: USINT;
END_VAR
(*выключаем все насосы кроме данного*)
FOR i := 1 TO MAX_K15_PUMPS_NUM DO
	IF i <> PumpID THEN
		fTurnOffK15Pump(i);
	END_IF;
END_FOR;

IF EmergencyPumpStopButtonPressed THEN	(*Нажат аварийный стоп насоса?*)
	fTurnOffK15Pump(PumpID); (*Выключить насос*)
	RETURN;
END_IF;

IF K15PumpFaulty[PumpID] THEN
	fTurnOffK15Pump(PumpID); (*Выключить насос*)
ELSE
	fTurnOnK15Pump(PumpID); (*Включить насос*)
END_IF;
END_FUNCTION

(* POU K16/fbK16PumpsControl, ST *)
FUNCTION_BLOCK fbK16PumpsControl
(*
	Управление насосами К16
	контура ГВС
*)
VAR CONSTANT
	PumpCheckDelayTime : TIME := T#10s;
	PumpWorkHeatingOrder : ARRAY [1..MAX_K16_PUMPS_NUM] OF USINT := 1, 2;
END_VAR
VAR_INPUT
	ManualMode: BOOL;						(*Ручной режим?*)
	WorkAllowed: BOOL;					(*Работа разрешена?*)
	EmergencyPumpStopButtonPressed: ARRAY [1..MAX_K16_PUMPS_NUM] OF BOOL; (*Нажат аварийный стоп насоса?*)
	PumpState: ARRAY [1..MAX_K16_PUMPS_NUM] OF BOOL;	(*Работает насос?*)
	PressureDrop : BOOL;					(*Есть разница давлений?*)
END_VAR
VAR_OUTPUT
END_VAR
VAR
	pumpStatusCheckDelay	: ARRAY [1..MAX_K16_PUMPS_NUM] OF TON;
	pumpsTrainingControl : fbK16PumpsTraining;
END_VAR

VAR_TEMP
	i : USINT;
	pumpWorkOrder : ARRAY [1..MAX_K16_PUMPS_NUM] OF USINT;
	pumpStatusCheck : ARRAY [1..MAX_K16_PUMPS_NUM] OF BOOL;
	break : BOOL := FALSE;
END_VAR
break := FALSE;

FOR i := 1 TO MAX_K16_PUMPS_NUM DO
	pumpStatusCheckDelay[i](IN := PumpState[i], PT := PumpCheckDelayTime);
	pumpStatusCheck[i] := pumpStatusCheckDelay[i].Q;
END_FOR;

fK16PumpsFaultyControl(
	PumpState				:= PumpState,
	PumpStatusCheckDelay	:= pumpStatusCheck,
	PressureDrop			:= PressureDrop
);

IF ManualMode THEN (*Ручной режим?*)
(*
	FOR i := 1 TO MAX_K16_PUMPS_NUM DO
		fK16PumpManualControl(
			PumpID	:= i,
			TurnOn	:= TurnOnPumpButtonPressed[i],
			TurnOff	:= TurnOffPumpButtonPressed[i],
			State		:= PumpState[i],
			EmergencyStop := EmergencyPumpStopButtonPressed[i]
		);
	END_FOR;
*)
	(*Контроллер никак не участвует в ручном режиме*)
	FOR i := 1 TO MAX_K16_PUMPS_NUM DO
		fTurnOffK16Pump(i);
	END_FOR;
ELSE
	IF WorkAllowed THEN	(*Работа разрешена?*)
		pumpWorkOrder := PumpWorkHeatingOrder;
		FOR i := 1 TO MAX_K16_PUMPS_NUM DO
			(*
				работаем с насосами в порядке их приоритета
				Ищем первый исправный насос и включаем его
			*)
			IF NOT(break) AND NOT(K16PumpFaulty[pumpWorkOrder[i]]) THEN
				fK16PumpAutoControl(
						PumpID := pumpWorkOrder[i],
						EmergencyPumpStopButtonPressed := EmergencyPumpStopButtonPressed[pumpWorkOrder[i]]
				);
				break := TRUE;
			END_IF;
		END_FOR;
		(*периодическая тренировка насосов*)
		pumpsTrainingControl();
	ELSE
		(*
			если работа не разрешена,
			выключаем все насосы
		*)
		FOR i := 1 TO MAX_K16_PUMPS_NUM DO
			fTurnOffK16Pump(i);
		END_FOR;
		RETURN;
	END_IF;
END_IF;
END_FUNCTION_BLOCK

(* POU K16/fbK16PumpsTraining, ST *)
FUNCTION_BLOCK fbK16PumpsTraining
(*
	Функция тренировки насосов К15
*)
VAR CONSTANT
	TrainingDelay: TIME := T#24h;		(*Задержка на включение тренировки*)
	TrainingPeriod: TIME := T#10s;	(*Период тренировки*)
END_VAR
VAR
	PumpOffDelay : ARRAY [1..MAX_K16_PUMPS_NUM] OF TON;
	PumpTrainingTimer : ARRAY [1..MAX_K16_PUMPS_NUM] OF TP;
END_VAR
VAR_TEMP
	i: USINT;
END_VAR
FOR i := 1 TO MAX_K16_PUMPS_NUM DO
	PumpOffDelay[i](IN := fGetK16Pump(i), PT := TrainingDelay);
	PumpTrainingTimer[i](IN := PumpOffDelay[i].Q, PT := TrainingPeriod);
	IF PumpTrainingTimer[i].Q THEN
		fTurnOnK16Pump(i);
	END_IF;
END_FOR;
END_FUNCTION_BLOCK

(* POU K16/fGetK16Pump, ST *)
FUNCTION fGetK16Pump :BOOL
(* Проверка включения насоса*)
VAR_INPUT
	PumpID : USINT;
END_VAR
fGetK16Pump := PLC160DO.K16Pump[PumpID];
END_FUNCTION

(* POU K16/fTurnOnK16Pump, ST *)
FUNCTION fTurnOnK16Pump : BOOL
VAR_INPUT
	PumpID : USINT;
END_VAR
fSetK16Pump(TRUE, PumpID);
END_FUNCTION

(* POU K16/fSetK16Pump, ST *)
FUNCTION fSetK16Pump : BOOL
VAR_INPUT
	State : BOOL;
	PumpID : USINT;
END_VAR
VAR
END_VAR
	PLC160DO.K16Pump[PumpID] := State;
	(*Включить/Выключить реле насоса*)
END_FUNCTION

(* POU K16/fK16PumpsFaultyControl, ST *)
FUNCTION fK16PumpsFaultyControl :BOOL
(* Проверка состояния насосов*)
VAR_INPUT
	PumpState : ARRAY [1..MAX_K16_PUMPS_NUM] OF BOOL;
	PumpStatusCheckDelay : ARRAY [1..MAX_K16_PUMPS_NUM] OF BOOL;
	PressureDrop : BOOL;
END_VAR
VAR
	i : USINT;
	activePumpID : USINT; (*номер работающего насоса*)
END_VAR
activePumpID := 0;

FOR i := 1 TO MAX_K16_PUMPS_NUM DO
	IF PumpState[i] THEN
		IF activePumpID <> 0 THEN
			(*
				Включено больше одного насоса -
				ничего не можем сказать об их исправности
			*)
			RETURN;
		END_IF;
		activePumpID := i;
	END_IF;
END_FOR;

IF activePumpID = 0 THEN
	(*
		Не включен ни один насос - 
		ничего не можем сказать об их исправности
	*)
	RETURN;
END_IF;

IF PumpStatusCheckDelay[activePumpID] THEN
	(*
		Определяем исправность насоса
		по перепаду давления
	*)
	K16PumpFaulty[activePumpID] := NOT(PressureDrop);
END_IF;
END_FUNCTION

(* POU K16/fTurnOffK16Pump, ST *)
FUNCTION fTurnOffK16Pump : BOOL
VAR_INPUT
	PumpID : USINT;
END_VAR
VAR
END_VAR
	fSetK16Pump(FALSE, PumpID);
END_FUNCTION

(* POU K16/fK16PumpAutoControl, ST *)
FUNCTION fK16PumpAutoControl : BOOL
VAR_INPUT
	PumpID : USINT;
	EmergencyPumpStopButtonPressed : BOOL;
END_VAR
VAR
	i: USINT;
END_VAR
(*выключаем все насосы кроме данного*)
FOR i := 1 TO MAX_K16_PUMPS_NUM DO
	IF i <> PumpID THEN
		fTurnOffK16Pump(i);
	END_IF;
END_FOR;

IF EmergencyPumpStopButtonPressed THEN	(*Нажат аварийный стоп насоса?*)
	fTurnOffK16Pump(PumpID); (*Выключить насос*)
	RETURN;
END_IF;

IF K16PumpFaulty[PumpID] THEN
	fTurnOffK16Pump(PumpID); (*Выключить насос*)
ELSE
	fTurnOnK16Pump(PumpID); (*Включить насос*)
END_IF;
END_FUNCTION

(* POU checkPumpsAlarm, ST *)
FUNCTION checkPumpsAlarm : BOOL
(*
	Включение лампочек и зуммера по авариям насосов
*)
VAR
	i : USINT;
END_VAR
	FOR i := 1 TO MAX_K14_PUMPS_NUM DO
		IF K14PumpFaulty[i] OR PLC160DI.UZStatus[i].Fail THEN
			MU110DO.K14PumpGroupAlarm := TRUE;
			MU110DO.Buzzer := TRUE;
		END_IF
	END_FOR;

	FOR i := 1 TO MAX_K15_PUMPS_NUM DO
		IF K15PumpFaulty[i] THEN
			PLC160DO.K15Alarm := TRUE;
			MU110DO.Buzzer := TRUE;
		END_IF
	END_FOR;

	FOR i := 1 TO MAX_K16_PUMPS_NUM DO
		IF K16PumpFaulty[i] THEN
			PLC160DO.K16Alarm := TRUE;
			MU110DO.Buzzer := TRUE;
		END_IF
	END_FOR;
END_FUNCTION

(* POU checkOtherAlarms, ST *)
FUNCTION checkOtherAlarms : BOOL
(*
	Включение зуммера по всяким другим авариям
*)
VAR
END_VAR
IF
	MV110DI.CO_Level_I	OR
	MV110DI.CO_Level_II	OR
	MV110DI.CH_Level_I	OR
	MV110DI.CH_Level_II	OR
	MV110DI.FireAlarm	OR
	MV110DI.BoilerGeneralFault	OR
	MV110DI.BoilerAlarm[1]	OR
	MV110DI.BoilerAlarm[2]	OR
	MV110DI.BoilerAlarm[3]	THEN
		MU110DO.Buzzer := TRUE;
END_IF
END_FUNCTION

(* POU resetPumpsAlarm, ST *)
FUNCTION resetPumpsAlarm : BOOL
(*
	Сброс всех аварий насосов
*)
VAR_INPUT
	IN : BOOL;
END_VAR
VAR
	i : USINT;
END_VAR
IF IN THEN
	MU110DO.K14PumpGroupAlarm := FALSE;
	PLC160DO.K15Alarm := FALSE;
	PLC160DO.K16Alarm := FALSE;
	MU110DO.Buzzer := FALSE;

	FOR i := 1 TO MAX_K14_PUMPS_NUM DO
		K14PumpFaulty[i] := FALSE;
	END_FOR;

	FOR i := 1 TO MAX_K15_PUMPS_NUM DO
		K15PumpFaulty[i] := FALSE;
	END_FOR;

	FOR i := 1 TO MAX_K16_PUMPS_NUM DO
		K16PumpFaulty[i] := FALSE;
	END_FOR;
END_IF;
END_FUNCTION

(* POU IO/GetInputs, ST *)
PROGRAM GetInputs
(*Дискртеные входы ПЛК160*)
PLC160DI.K14_PumpsModeIsAuto		:= DI_0_00;
PLC160DI.K14_PumpsModeIsHeating	:= NOT(DI_0_01);
PLC160DI.K14_PumpStop[1]			:= DI_0_02;
PLC160DI.K14_PumpStop[2]			:= DI_0_03;
PLC160DI.K14_PumpStop[3]			:= DI_0_04;
PLC160DI.K14_NoPressureDrop		:= DI_0_05;
PLC160DI.UZStatus[1].Ready			:= DI_0_06;
PLC160DI.UZStatus[1].Running		:= DI_0_07;
PLC160DI.UZStatus[1].Fail			:= NOT(DI_0_08);
PLC160DI.UZStatus[2].Ready			:= DI_0_09;
PLC160DI.UZStatus[2].Running		:= DI_0_10;
PLC160DI.UZStatus[2].Fail			:= NOT(DI_0_11);
PLC160DI.UZStatus[3].Ready			:= DI_0_12;
PLC160DI.UZStatus[3].Running		:= DI_0_13;
PLC160DI.UZStatus[3].Fail			:= NOT(DI_0_14);
PLC160DI.Reserved						:= DI_0_15;

(*Аналоговые входы ПЛК160*)
PLC160AI.UZSignal[1]					:= AI_0_00;
PLC160AI.UZSignal[2]					:= AI_0_01;
PLC160AI.UZSignal[3]					:= AI_0_02;
PLC160AI.DilutionSignal[1]			:= AI_0_03;
PLC160AI.DilutionSignal[2]			:= AI_0_04;
PLC160AI.DilutionSignal[3]			:= AI_0_05;
PLC160AI.Reserved[1]					:= AI_0_06;
PLC160AI.Reserved[2]					:= AI_0_07;

(*Дискретные входы МВ110-ДН32*)
MV110DI.K15_StopButton[1]			:= getMV110Input(0);
MV110DI.K15_StopButton[2]			:= getMV110Input(1);
MV110DI.K16_StopButton[1]			:= getMV110Input(2);
MV110DI.K16_StopButton[2]			:= getMV110Input(3);
MV110DI.K15_NoPressureDrop			:= getMV110Input(4);
MV110DI.K16_NoPressureDrop			:= getMV110Input(5);
MV110DI.HeatingDHWPumpGroupModeIsAuto	:= getMV110Input(6);
MV110DI.DHWPumpGroupModeIsAuto	:= getMV110Input(7);
MV110DI.CO_Level_I					:= getMV110Input(8);
MV110DI.CO_Level_II					:= getMV110Input(9);
MV110DI.CH_Level_I					:= getMV110Input(10);
MV110DI.CH_Level_II					:= getMV110Input(11);
MV110DI.FireAlarm						:= getMV110Input(12);
MV110DI.BoilerGeneralFault			:= getMV110Input(13);
MV110DI.TurnOnK15AndK16				:= getMV110Input(14);
MV110DI.K22ValveState.Open			:= getMV110Input(15);
MV110DI.K22ValveState.Close		:= getMV110Input(16);
MV110DI.K23ValveState.Open			:= getMV110Input(17);
MV110DI.K23ValveState.Close		:= getMV110Input(18);
MV110DI.BoilerAlarm[1]				:= getMV110Input(19);
MV110DI.BoilerAlarm[2]				:= getMV110Input(20);
MV110DI.BoilerAlarm[3]				:= getMV110Input(21);
MV110DI.BlockAllBoilers				:= getMV110Input(22);
MV110DI.TurnOnAllBoilers			:= getMV110Input(23);
MV110DI.SignalizationButton		:= getMV110Input(24);
MV110DI.QFSwitcher[1]				:= getMV110Input(25);
MV110DI.QFSwitcher[2]				:= getMV110Input(26);
MV110DI.QFSwitcher[3]				:= getMV110Input(27);
MV110DI.QFSwitcher[4]				:= getMV110Input(28);
MV110DI.QFSwitcher[5]				:= getMV110Input(29);
MV110DI.QFSwitcher[6]				:= getMV110Input(30);
MV110DI.QFSwitcher[7]				:= getMV110Input(31);
END_PROGRAM

(* POU IO/getMV110Input, ST *)
FUNCTION getMV110Input : BOOL
VAR_INPUT
	IN : USINT;
END_VAR
VAR
END_VAR
getMV110Input := EXTRACT(DI_1, IN);
END_FUNCTION

(* POU IO/SetOutputs, ST *)
PROGRAM SetOutputs
VAR
END_VAR
(*Аналоговые выходы ПЛК160*)
AO_0_00 := PLC160AO.UZSpeed[1];
AO_0_01 := PLC160AO.UZSpeed[2];
AO_0_02 := PLC160AO.UZSpeed[3];
AO_0_03 := PLC160AO.Reserved;

(*Дискретные выходы ПЛК160*)
DO_0_00 := PLC160DO.UZStart[1];
DO_0_01 := PLC160DO.UZStart[2];
DO_0_02 := PLC160DO.UZStart[3];
DO_0_03 := PLC160DO.UZConstSpeed[1];
DO_0_04 := PLC160DO.UZConstSpeed[2];
DO_0_05 := PLC160DO.UZConstSpeed[3];
DO_0_06 := PLC160DO.K15Pump[1];
DO_0_07 := PLC160DO.K15Pump[2];
DO_0_08 := PLC160DO.K16Pump[1];
DO_0_09 := PLC160DO.K16Pump[2];
DO_0_10 := PLC160DO.K15Alarm;
DO_0_11 := PLC160DO.K16Alarm;

(*Дискретные выходы МУ110-8Р*)
DO_1_00 := setMUOutput(MU110DO.K14PumpGroupAlarm);
DO_1_01 := setMUOutput(MU110DO.Buzzer);
DO_1_02 := setMUOutput(MU110DO.K14PumpIsOn[1]);
DO_1_03 := setMUOutput(MU110DO.K14PumpIsOn[2]);
DO_1_04 := setMUOutput(MU110DO.K14PumpIsOn[3]);
DO_1_05 := setMUOutput(MU110DO.Reserved[1]);
DO_1_06 := setMUOutput(MU110DO.Reserved[2]);
DO_1_07 := setMUOutput(MU110DO.Reserved[3]);
END_PROGRAM

(* POU IO/setMUOutput, ST *)
FUNCTION setMUOutput : WORD
VAR_INPUT
	IN : BOOL;
END_VAR
VAR
END_VAR
IF IN THEN
	setMUOutput := 1000;
ELSE
	setMUOutput := 0;
END_IF;
END_FUNCTION

(* POU K14/fK14PumpManualControl, ST *)
FUNCTION fK14PumpManualControl : BOOL
VAR_INPUT
	PumpID : USINT;
	TurnOn : BOOL;
	TurnOff : BOOL;
	State : BOOL;
	EmergencyStop : BOOL;
END_VAR
VAR
END_VAR
IF TurnOn OR State THEN (*Нажата кнопка "Пуск насоса" или Работает насос?*)
	IF TurnOff THEN (*Нажата кнопка "Стоп насоса"?*)
		fTurnOffK14Pump(PumpID);
		RETURN;
	ELSE
		IF EmergencyStop THEN (*Нажат аварийный стоп насоса?*)
			fTurnOffK14Pump(PumpID);
			RETURN;
		ELSE
			fTurnOnK14Pump(PumpID);
			RETURN;
		END_IF;
	END_IF;
ELSE
	RETURN;
END_IF;
END_FUNCTION

(* POU K15/fK15PumpManualControl, ST *)
FUNCTION fK15PumpManualControl : BOOL
VAR_INPUT
	PumpID : USINT;
	TurnOn : BOOL;
	TurnOff : BOOL;
	State : BOOL;
	EmergencyStop : BOOL;
END_VAR
VAR
END_VAR
IF TurnOn OR State THEN (*Нажата кнопка "Пуск насоса" или Работает насос?*)
	IF TurnOff THEN (*Нажата кнопка "Стоп насоса"?*)
		fTurnOffK15Pump(PumpID);
		RETURN;
	ELSE
		IF EmergencyStop THEN (*Нажат аварийный стоп насоса?*)
			fTurnOffK15Pump(PumpID);
			RETURN;
		ELSE
			fTurnOnK15Pump(PumpID);
			RETURN;
		END_IF;
	END_IF;
ELSE
	RETURN;
END_IF;
END_FUNCTION

(* POU K16/fK16PumpManualControl, ST *)
FUNCTION fK16PumpManualControl : BOOL
VAR_INPUT
	PumpID : USINT;
	TurnOn : BOOL;
	TurnOff : BOOL;
	State : BOOL;
	EmergencyStop : BOOL;
END_VAR
VAR
END_VAR
IF TurnOn OR State THEN (*Нажата кнопка "Пуск насоса" или Работает насос?*)
	IF TurnOff THEN (*Нажата кнопка "Стоп насоса"?*)
		fTurnOffK16Pump(PumpID);
		RETURN;
	ELSE
		IF EmergencyStop THEN (*Нажат аварийный стоп насоса?*)
			fTurnOffK16Pump(PumpID);
			RETURN;
		ELSE
			fTurnOnK16Pump(PumpID);
			RETURN;
		END_IF;
	END_IF;
ELSE
	RETURN;
END_IF;
END_FUNCTION
